FUNCTION_BLOCK FB_Subject IMPLEMENTS InterfaceEventViewer
VAR CONSTANT
	MAX_EVENTS : UDINT := 10;
END_VAR
VAR
	event_containers	: ARRAY [1..MAX_EVENTS] OF InterfaceEventViewer;
	max_index			: UDINT;
END_VAR

{warning 'add method implementation '}
METHOD clear : BOOL
VAR
	i : UDINT;
END_VAR
FOR i := 1 TO max_index DO
	IF event_containers[i] <> 0 THEN
		event_containers[i].clear();
	END_IF
END_FOR
END_METHOD

{warning 'add method implementation '}
METHOD history_clear : BOOL
VAR
	i : UDINT;
END_VAR
FOR i := 1 TO max_index DO
	IF event_containers[i] <> 0 THEN
		event_containers[i].history_clear();
	END_IF
END_FOR
END_METHOD

{warning 'add method implementation '}
METHOD send_event : BOOL
VAR_INPUT
	event_container	: REFERENCE TO EventContainer;
END_VAR
VAR
	i : UDINT;
END_VAR
FOR i := 1 TO max_index DO
	IF event_containers[i] <> 0 THEN
		event_containers[i].send_event(event_container);
	END_IF
END_FOR
END_METHOD

{warning 'add method implementation '}
METHOD show : BOOL
VAR_INPUT
	event_container	: REFERENCE TO EventContainer;
END_VAR
VAR
	i : UDINT;
END_VAR
FOR i := 1 TO max_index DO
	IF event_containers[i] <> 0 THEN
		event_containers[i].show(event_container);
	END_IF
END_FOR
END_METHOD

METHOD subscribe : UDINT
VAR_INPUT
	observable	: InterfaceEventViewer;
END_VAR
VAR
	i : UDINT;
END_VAR
subscribe := 0;
FOR i := 1 TO MAX_EVENTS DO
	IF event_containers[i] = 0 THEN
		event_containers[i] := observable;
		IF i > max_index THEN
			max_index := i;
		END_IF
		subscribe := i;
		RETURN;
	END_IF
END_FOR
END_METHOD

METHOD unsubscribe : BOOL
VAR_INPUT
	subscriber : UDINT;
END_VAR
VAR
	i : UDINT;
END_VAR
IF event_containers[subscriber] <> 0 THEN
	event_containers[subscriber] := 0;
	IF subscriber = max_index THEN
		FOR i := max_index TO 0 BY -1 DO
			IF event_containers[i] <> 0 THEN
				max_index := 1;
			END_IF
		END_FOR
	END_IF
	unsubscribe := TRUE;
ELSE
	unsubscribe := FALSE;
END_IF
END_METHOD

END_FUNCTION_BLOCK

(* stored: Version 1.1.0.1, ProductVersion 3.1.4024.15
   POU FB_Subject: Id {6ed8c9cd-86ba-4ebc-ba32-2dcbc2e1f434}, SpecialFunc None
   Method clear: Id {580ee6da-d3b7-42e4-898e-f42aa81df34e}
   Method history_clear: Id {6cfa058d-9ed8-4cb2-b7af-8a6728d3c7d9}
   Method send_event: Id {6c7126ec-fc35-4109-87ac-3644d2cc1d03}
   Method show: Id {4bba132d-4ddc-4512-9240-4527f3c06f89}
   Method subscribe: Id {84e41b96-1fc0-4513-9b69-b0b5199d83a0}
   Method unsubscribe: Id {0f0923f2-7ad9-4d02-8ee4-ac2ac38832ed} *)
